INTERFACE Temp_ITFPalletPins

METHOD Beweegpinsnaarbeneden
VAR_INPUT
END_VAR
END_METHOD

METHOD ErinBewegen
VAR_INPUT
END_VAR
END_METHOD

METHOD EruitBewegen
VAR_INPUT
END_VAR
END_METHOD

END_INTERFACE

(* stored: Version 1.1.0.1
   Itf Temp_ITFPalletPins: Id {b3648339-c988-4d5f-97cd-8a7fdd9c6865}
   Method Beweegpinsnaarbeneden: Id {82450bbc-49b3-4bf2-b6bf-e632ecb152d1}
   Method ErinBewegen: Id {57139f31-177b-4f4d-892d-369d551493be}
   Method EruitBewegen: Id {556d00d9-3f23-492c-80b0-4ea7920c6b24} *)
